TYPE FB_httpClient_State :
(
	UNDEFINIERT := 0,
	GETRENNT,
	VERBUNDEN,
	SENDEN,
	ANTWORT_ERFASSEN,
	ANTWORT_AUSWERTEN,
	
	
	ERROR_HANDLER
);
END_TYPE

(* stored: Version 1.1.0.1, ProductVersion 3.1.4018.5
   DUT FB_httpClient_State: Id {debf35aa-b43c-4f11-920f-f1a076920e41} *)
